(* PLC project robotctrl, Dassault Systèmes ControlBuild 2024x Refresh1 *)
(* stored: creationDateTime 2024-04-17T16:28:53-01:00 *)

FUNCTION_BLOCK flask_motion_app.robotctrl
  VAR_INPUT
    forwardUp : BOOL := false;
    backwardUp : BOOL := false;
  END_VAR
  VAR_INPUT
    forwardDw : BOOL := false;
    backwardDw : BOOL := false;
  END_VAR
  VAR_INPUT
    presConvUp : BOOL := false;
    presConvDw : BOOL := false;
    masterPosition : REAL := 0.0;
  END_VAR
  VAR_INPUT
    Auto : BOOL := false;
    Manu : BOOL := false;
    run : BOOL := false;
  END_VAR
  VAR_INPUT
    weightOk : BOOL := false;
  END_VAR
  VAR_OUTPUT
    phaseCode : INT := 0;
  END_VAR
  VAR_OUTPUT
    HomeCmd : BOOL := false;
    MoveVelCmd : BOOL := false;
    MoveAbsCmd : BOOL := false;
    MoveVel1ManualCmd : BOOL := false;
    MoveVel2ManualCmd : BOOL := false;
    MoveAbs1ManualCmd : BOOL := false;
    MoveAbs2ManualCmd : BOOL := false;
    StopCmd : BOOL := false;
    MovePosition : REAL := 0.0;
    MoveSpeed : REAL := 100.0;
    MoveAcceleration : REAL := 100.0;
    MoveDeceleration : REAL := 100.0;
    offsetAxToMa : REAL := 0.0;
    gripSyringes : BOOL := false;
  END_VAR
  VAR CONSTANT
    endPhase1 : REAL := 50.0;
    endPhase2 : REAL := 60.0;
    endPhase3 : REAL := 150.0;
    endPhase4 : REAL := 200.0;
    speedPhase1 : REAL := 80.0;
    speedPhase2 : REAL := 85.0;
    speedPhase3 : REAL := 100.0;
    speedPhase4 : REAL := 100.0;
    globalSpeedFactor : REAL := 100.0;
  END_VAR

(* comment *)
(* comment *)
(* comment *)
(* comment *)

if ((masterPosition >=0.0) and (masterPosition < endPhase1 )) then phaseCode := 1; end_if;
if ((masterPosition >= endPhase1 ) and (masterPosition <endPhase2)) then phaseCode := 2; end_if;
if ((masterPosition >= endPhase2 ) and (masterPosition <endPhase3)) then phaseCode := 3; end_if;
if ((masterPosition >= endPhase3 ) and (masterPosition <endPhase4)) then phaseCode := 4; end_if;
if ((masterPosition >= endPhase4 ) and (masterPosition <360.0)) then phaseCode := 5; end_if;

if ((phaseCode = 2) and (not presConvDw or not weightOk)) then phaseCode := 0; end_if;
if ((phaseCode = 3) and presConvUp) then phaseCode := 0; end_if;
if (not run) then  phaseCode := 0; end_if;

CASE phaseCode OF
	0: 	MoveVelCmd := false;


	1 : 	MoveVelCmd := true ;  (* Approach to take the product *)
		MoveSpeed := speedPhase1 * globalSpeedFactor /100.0 ;
		gripSyringes := false;
		
	2 :	MoveVelCmd := true ;	(* take the product slowly *)
		MoveSpeed := speedPhase2 * globalSpeedFactor /100.0 ;
		gripSyringes := true;

	3 :	MoveVelCmd := true ;	(* Go the the second conveyor *)
		MoveSpeed := speedPhase3 * globalSpeedFactor /100.0 ;
		gripSyringes := true;

	4 :	MoveVelCmd := true ;	(* put down the product *)
		MoveSpeed := speedPhase4 * globalSpeedFactor /100.0 ; 	
		gripSyringes := true;
	
	5 :	MoveVelCmd := true ;	(* go back *)
		MoveSpeed := speedPhase4 * globalSpeedFactor /100.0 ; 	
		gripSyringes := false;

ELSE 	
	MoveVelCmd := false ;
	
END_CASE;
END_FUNCTION_BLOCK
